{attribute 'qualified_only'}
{attribute 'strict'}
TYPE ENUM_StationCommand :
(
  	
    INIT :=1,
    START := 2,
    STOP :=3,
    PAUSE := 4
    
    
  
);
END_TYPE

(* stored: Version 1.1.0.1, ProductVersion 3.1.4024.12
   DUT ENUM_StationCommand: Id {134f1a16-2527-4649-86a0-9fd29189cfd4} *)
